FUNCTION_BLOCK FB_OdometryOpponents
VAR_INPUT
END_VAR
VAR_OUTPUT
END_VAR
VAR
END_VAR

END_FUNCTION_BLOCK

(* stored: Version 1.1.0.1, ProductVersion 3.1.4022.18
   POU FB_OdometryOpponents: Id {b0c0ab87-41b9-4d27-8187-f433cf8bb0e9}, SpecialFunc None *)
